INTERFACE INTERNAL I_JobInternal EXTENDS I_Debug

PROPERTY INTERNAL _Next : I_Job
GET
END_GET
SET
END_SET
END_PROPERTY

METHOD INTERNAL _OnAbort
VAR_INPUT
END_VAR
END_METHOD

METHOD INTERNAL _OnDone
VAR_INPUT
END_VAR
END_METHOD

METHOD INTERNAL _OnExit
VAR_INPUT
END_VAR
END_METHOD

METHOD INTERNAL _OnRun
VAR_INPUT
END_VAR
END_METHOD

METHOD INTERNAL _OnStart
VAR_INPUT
END_VAR
END_METHOD

PROPERTY INTERNAL _Prev : I_Job
GET
END_GET
SET
END_SET
END_PROPERTY

(*
Returns Jobs state
*)
PROPERTY State : JobState
GET
END_GET
END_PROPERTY

(*
Returns Worker working on this job
*)
PROPERTY Worker : I_Worker
GET
END_GET
END_PROPERTY

END_INTERFACE

(* stored: Version 1.1.0.1
   Itf I_JobInternal: Id {2ce45242-2ee2-48fc-8798-89f355749e56}
   Property _Next: Id {87fef1e3-f6f6-46a4-b39e-7c0b718fd672}
   Get Get: Id {2d0ace25-2d9c-4ce3-a2c5-ea616c65d679}
   Set Set: Id {4e927b31-f06b-4ab1-a402-ebcc7ca91a3c}
   Method _OnAbort: Id {40811cca-b370-45e3-ba69-091549bb0e7e}
   Method _OnDone: Id {fd4b7884-d760-484c-b0b2-935bdb12e0bd}
   Method _OnExit: Id {d60c12a1-ac1b-48e0-93bd-01ab51aa13b1}
   Method _OnRun: Id {e7f78728-5390-480e-8201-6cfd17b69308}
   Method _OnStart: Id {7c415d3b-2b45-4c1c-8877-d685d666638d}
   Property _Prev: Id {dd5d9bdd-695b-471b-8165-18c58991ba5f}
   Get Get: Id {bb9f53b5-605e-454a-b1c0-4ff5189e2dea}
   Set Set: Id {cfc6a368-ef90-45f9-8ff0-40461c10d82c}
   Property State: Id {40ba106d-f5cb-44d4-93ab-1d5747fe9c61}
   Get Get: Id {47eba237-e8ec-4d0a-98fa-6628f9e6e51e}
   Property Worker: Id {ebd0c1e4-e352-4924-86df-3b078a72350c}
   Get Get: Id {9cd67c7f-916b-4d21-9b45-6dd0590dadaf} *)
